{attribute 'linkalways'} 
{attribute 'no_explicit_call' := 'This FB is a CLASS and must be accessed using methods or properties'}
{attribute 'enable_dynamic_creation'}
FUNCTION_BLOCK ABSTRACT LinkedListEvent EXTENDS Disposable
VAR
	_targetLinkedList : I_LinkedList;
END_VAR

METHOD FB_init : BOOL
VAR_INPUT
	bInitRetains : BOOL; // if TRUE, the retain variables are initialized (warm start / cold start)
	bInCopyCode : BOOL;  // if TRUE, the instance afterwards gets moved into the copy code (online change)
	TargetLinkedList : I_LinkedList;
END_VAR
THIS^._targetLinkedList := TargetLinkedList;
END_METHOD

PROPERTY PUBLIC TargetLinkedList : I_LinkedList
GET // PUBLIC
TargetLinkedList := _targetLinkedList;
END_GET
END_PROPERTY

END_FUNCTION_BLOCK

(* stored: Version 1.1.0.1, ProductVersion 3.1.4024.12
   POU LinkedListEvent: Id {96cbd876-2741-4b0f-bb8e-9e022ea8faf2}, SpecialFunc None
   Folder Constructor: Id {193d9d60-21dd-4461-a8bf-915d0e152d0f}
   Method FB_init: Id {06bb3ad0-ab29-4387-8693-b12f3f386d17}
   Property TargetLinkedList: Id {c3047d9f-5588-4093-8c28-b7a126bcc0c0}
   Get Get: Id {10549787-9390-4a77-9f43-0182fe39840d} *)
